FUNCTION_BLOCK FB_piec
VAR_INPUT
END_VAR
VAR_OUTPUT
END_VAR
VAR
    stan:INT ;
    pozycjaWzdluz:INT ;
    pozycjaHoruzontalna:INT ;	
END_VAR

CASE stan OF
    0:
        IF pozycjaWzdluz<430 THEN
            pozycjaWzdluz:=pozycjaWzdluz +1;
        END_IF
        IF pozycjaWzdluz=430 THEN
            stan:=1;
        END_IF
    1:
        IF pozycjaHoruzontalna<110 THEN
            pozycjaHoruzontalna:=pozycjaHoruzontalna +1;
        END_IF
        IF pozycjaHoruzontalna = 110 THEN
            stan:=3;
        END_IF
    2:
        IF pozycjaWzdluz < 650 THEN
            pozycjaWzdluz:=pozycjaWzdluz +1;
        END_IF
        IF pozycjaWzdluz = 650 THEN
            stan:=3;
        END_IF
    3:
        metoda_Restart();

END_CASE

METHOD metoda_Restart : BOOL
VAR_INPUT
END_VAR
pozycjaWzdluz :=0;
pozycjaHoruzontalna :=0;
stan :=0;
END_METHOD

END_FUNCTION_BLOCK

(* stored: Version 1.1.0.1, ProductVersion 3.1.4024.4
   POU FB_piec: Id {a93a0b2e-5986-4e06-b667-625518369fa2}, SpecialFunc None
   Method metoda_Restart: Id {d17195e1-c8c8-46a7-ac62-ff5c67235533} *)
